// TwinCAT 3 PLC project PLC01
// ProgramVersion: 3.1.4024.0
// libraries:
//   Tc2_Standard, * (Beckhoff Automation GmbH)
//   Tc2_System, * (Beckhoff Automation GmbH)
//   Tc2_Utilities, * (Beckhoff Automation GmbH)
//   Tc3_Module, * (Beckhoff Automation GmbH)
// project tree:
//   DUTs/ E_EventType.TcDUT (not stored), st_Event.TcDUT (not stored)
//   / PlcTask.TcTTO (not stored)
//   POUs/ Class Diagram.TcCD (not stored), EventLogger.TcPOU, FB_Rectangle.TcPOU (not stored), FB_RectangleChild.TcPOU, I_Shape.TcIO (not stored), MAIN.TcPOU, UpdateEventTimeStampSystemTime.TcPOU

// ---- POUs/EventLogger.TcPOU
FUNCTION_BLOCK EventLogger
VAR
	EventBuffer : ARRAY{1..TamanhoBuffer} OF st_Event;
	EventBufferID : INT := 0;
END_VAR
VAR CONSTANT
	TamanhoBuffer : INT := 100;
END_VAR

// Retorna verdadeiro se adição de evento foi concluída, falso se o buffer está cheio
METHOD PUBLIC AddEvent : BOOL
VAR_INPUT
	eEventType : E_EventType;
	eEventSeverity : TcEventSeverity;
	nEventIdentity : UDINT;
	sEventText : STRING(255);
END_VAR
IF NOT BufferCheio() THEN
	// Sem código ainda
	EventBufferID := EventBufferID + 1;
	EventBuffer[]
	AddEvent := TRUE;
ELSE
	AddEvent := FALSE;
END_IF
END_METHOD

METHOD PRIVATE BufferCheio : BOOL
IF (EventBufferID + 1) > TamanhoBuffer THEN
	BufferCheio := TRUE;
ELSE
	BufferCheio := FALSE;
END_IF
END_METHOD

END_FUNCTION_BLOCK

// ---- POUs/FB_RectangleChild.TcPOU
FUNCTION_BLOCK FB_RectangleChild EXTENDS FB_Rectangle
VAR_INPUT
END_VAR
VAR_OUTPUT
END_VAR
VAR
END_VAR

END_FUNCTION_BLOCK

// ---- POUs/MAIN.TcPOU
PROGRAM MAIN
VAR
	stInstance : st_Event;
	bBoolean : BOOL := FALSE;
	RectangleA : FB_Rectangle;
	RectangleB : FB_Rectangle;
END_VAR

IF NOT bBoolean THEN
	UpdateEventTimeStampSystemTime (stEvent := stInstance);
	bBoolean := TRUE;
END_IF

END_PROGRAM

// ---- POUs/UpdateEventTimeStampSystemTime.TcPOU
FUNCTION UpdateEventTimeStampSystemTime
VAR_INPUT
	stEvent : REFERENCE TO ST_Event;
END_VAR
VAR
	fbGETSYSTEMTIME : GETSYSTEMTIME;
	stFileTime : T_FILETIME;
END_VAR

fbGETSYSTEMTIME (TimeLoDW => stFileTime.dwLowDateTime,
				TimeHiDW => stFileTime.dwHighDateTime);

stEvent.dtTimeStamp := FILETIME_TO_DT (fileTime := stFileTime);

END_FUNCTION
